{attribute addProperty BoxType "AMP8000-0000-0103-0103"}
{attribute addProperty Id "AdsAddrAT %I*AMSADDR6480DcOutputShiftAT %I*DINT3240DcInputShiftAT %I*DINT3240AoeNetIdAT %I*AMSNETID4860Chn0AT %I*USINT810StateAT %I*UINT1620"}
{attribute addProperty CRC "4029734043"}
{attribute addProperty SizeInBites "200"}
{attribute addProperty SizeInBytes "25"}
TYPE InfoData_F030DC9B :
STRUCT
	{attribute addProperty Name "AdsAddr"}
	AdsAddr AT %I* : AMSADDR;
	{attribute addProperty Name "DcOutputShift"}
	DcOutputShift AT %I* : DINT;
	{attribute addProperty Name "DcInputShift"}
	DcInputShift AT %I* : DINT;
	{attribute addProperty Name "AoeNetId"}
	AoeNetId AT %I* : AMSNETID;
	{attribute addProperty Name "Chn0"}
	Chn0 AT %I* : USINT;
	{attribute addProperty Name "State"}
	State AT %I* : UINT;
END_STRUCT
END_TYPE

(* stored: Version 1.2.0.0, ProductVersion 3.1.4024.9
   DUT InfoData_F030DC9B: Id {09ce723b-2944-456e-9b7a-9fea57367dc2} *)
